{attribute 'qualified_only'}
VAR_GLOBAL
	nDALILine				:	INT := 1; // Start with DALI-Line 1 as default.
END_VAR
VAR_GLOBAL CONSTANT
	nNumberOfDALI_Lines		: 	INT := 10; // Constant to vary with the number of required DALI Lines.
END_VAR

(* stored: Version 1.1.0.1, ProductVersion 3.1.4024.10
   GVL GVL_Internal: Id {5c8f73e6-ddca-4782-8329-aa5c5ce707a2} *)
